PROGRAM Reset
(*What happens when reset is pressed*)
VAR
END_VAR

IF GVL.Reset_Count THEN
	GVL.ProductA_Amount := 0; (*To Reset Product Count*)
	GVL.ProductB_Amount := 0; (*To Reset Product Count*)
END_IF

END_PROGRAM

(* stored: Version 1.1.0.1, ProductVersion 3.1.4024.12
   POU Reset: Id {508545e5-b58e-408c-98c8-3800502ff6ab}, SpecialFunc None *)
